/// Data of one tracking window
TYPE ST_WindowTrackingWindow :
(************************************************************************************** 
* 	Application 		: BoxControl Framework 
* 	Revision 			: $Revision: 408723 $ 
* 	Revision date 		: $Date: 2018-06-27 13:49:08 +0200 (Wed, 27 Jun 2018) $ 
* 	Last changed by 	: $Author: b7bolm $ 
* 	URL 				: $URL: http://almscdc.swisslog.com/repo/SWPD/Development/BoxControlFramework/21_Projects/BCF_2.0/trunk/BCF/BCF/JumpStart/20_Product/10_App/12_E_Functions/10_Lib/10_Conv/FB_FunctionList.TcPOU $ 
* ------------------------------------------------------------------------------------ 
* 	© Swisslog AG 
* 	Swisslog is not liable for any usage of this source code that is not agreed 
* 	on between Swisslog and the other party. The mandatory legal liability remains 
* 	unaffected. 
* ------------------------------------------------------------------------------------ 
* 	Revision History: 
* 
* 	VERSION 		DATE 			INITIALS 			DESCRIPTION 
* 	0.1 			24.08.2018 		ahe 				First implementation
* 
**************************************************************************************)
STRUCT
	TU_FrontEdgePosition	: UDINT;
	TU_RearEdgePosition		: UDINT;
	State					: E_WindowTrackingWindowState;
	ZoneIndex				: UINT;
	Flush					: BOOL;
END_STRUCT
END_TYPE

(* stored: Version 1.1.0.1, ProductVersion 3.1.4020.6
   DUT ST_WindowTrackingWindow: Id {ce3148a1-87b4-4ae1-9049-b1ef1e104b45} *)
